{attribute 'GeneratedUsingTerminal: EL5101-0000-0001'}
{attribute addProperty BoxType "EL5101-0000-0001"}
{attribute addProperty Id "CtrlAT %Q*USINT1ValueAT %Q*UINT2"}
{attribute addProperty CRC "3329760021"}
{attribute addProperty Size "3"}
TYPE Outputs_C6781B15 :
STRUCT
	{attribute addProperty Name "Ctrl"}
	Ctrl AT %Q* : USINT;
	{attribute addProperty Name "Value"}
	Value AT %Q* : UINT;
END_STRUCT
END_TYPE

(* stored: Version 1.2.0.0, ProductVersion 3.1.4024.9
   DUT Outputs_C6781B15: Id {a9b89fe9-3d7d-4241-b558-2796648b12df} *)
